Fanuc KAREL source: kc00042.KL

-- PROVISIONAL review KL for V940-1; original PC SHA256 ac2bc3e96b4922acab0ce398e6e0a871b346be38e1f5a41425f43b4e801f78cf
-- Incomplete behavior may be omitted. Consult companion uncertainty JSON. Do not deploy.
PROGRAM KC00042
%NOLOCKGROUP
BEGIN
  -- V9_ZERO_TABLE_METADATA_HINT layout=0002_ascii; no indexed target words; source/name/runtime held
  -- UNRESOLVED_PC offsets 5-35; opcodes 27,22,22,27,9D,31,7E,4A
  -- UNRESOLVED_PC offsets 40-44; opcodes 7F
END KC00042
